(* PLC project Unnamed, Unknown Unnamed 1 *)
(* stored: creationDateTime 2023-01-31T01:35:27, modificationDateTime 2023-04-25T02:26:45 *)

PROGRAM WaterIrrigation
  VAR
    OUTGOING_VALVE AT %QX0.0 : BOOL;
    OUTGOING_PUMP AT %QX0.1 : BOOL;
    INCOMING_PUMP AT %QX0.2 : BOOL;
    TANK_FULL AT %QX0.3 : BOOL;
    PULSE AT %QX0.4 : BOOL;
    TANK_EMPTY AT %QX0.5 : BOOL;
    MANUAL AT %QX0.6 : BOOL;
    PB_INCOMING_OPEN AT %IX0.0 : BOOL;
    PB_INCOMING_CLOSE AT %IX0.1 : BOOL;
    PB_OUTGOING_OPEN AT %IX0.2 : BOOL;
    PB_OUTGOING_CLOSE AT %IX0.3 : BOOL;
    MAX_TANK_LEVEL AT %QW0 : INT := 10;
    TANK_LEVEL_VALUE AT %QW2 : INT := 10;
    WATER_MOISTURE AT %QW3 : INT := 10;
  END_VAR
  VAR
    TON0 : TON;
    TOF0 : TOF;
    CTUD0 : CTUD;
  END_VAR
  VAR  (* added by the conversion: wires and edge detectors of the diagram *)
    R_TRIG1 : R_TRIG;
    R_TRIG2 : R_TRIG;
  END_VAR

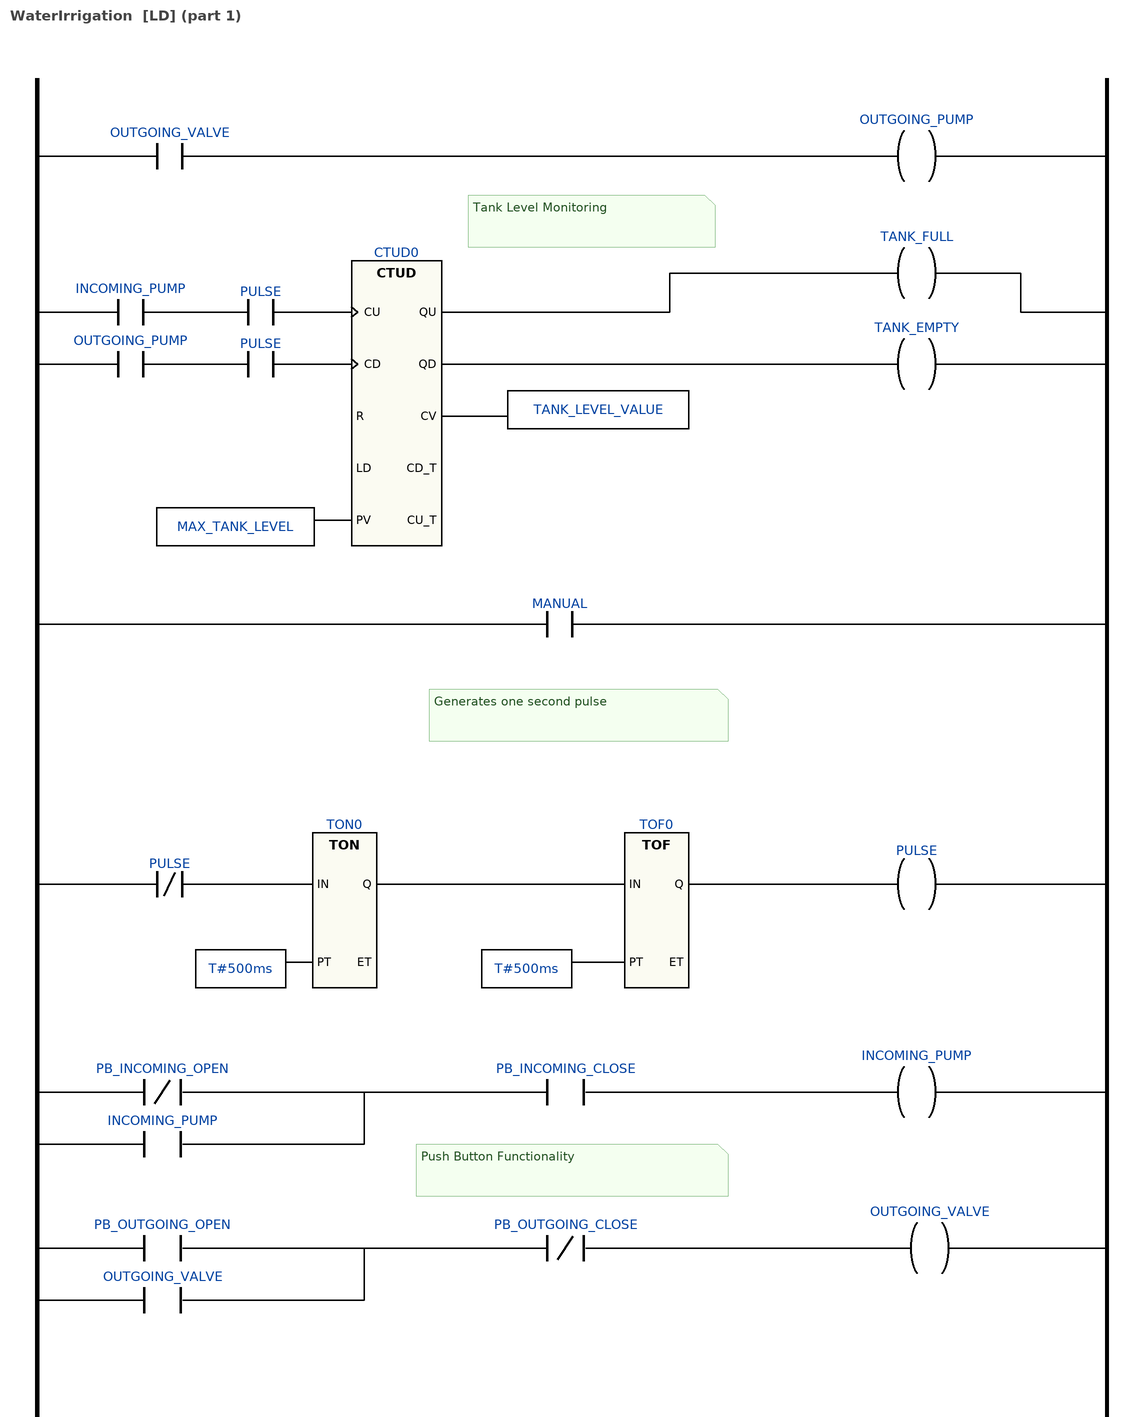
(* LD diagram, written out as Structured Text *)
OUTGOING_PUMP := OUTGOING_VALVE;
(* Tank Level Monitoring *)
R_TRIG1(CLK := INCOMING_PUMP AND PULSE);
R_TRIG2(CLK := OUTGOING_PUMP AND PULSE);
CTUD0(CU := R_TRIG1.Q, CD := R_TRIG2.Q, PV := MAX_TANK_LEVEL);
TANK_FULL := CTUD0.QU;
TANK_EMPTY := CTUD0.QD;
TANK_LEVEL_VALUE := CTUD0.CV;
(* Generates one second pulse *)
TON0(IN := NOT PULSE, PT := T#500ms);
TOF0(IN := TON0.Q, PT := T#500ms);
PULSE := TOF0.Q;
INCOMING_PUMP := (NOT PB_INCOMING_OPEN OR INCOMING_PUMP) AND PB_INCOMING_CLOSE;
(* Push Button Functionality *)
OUTGOING_VALVE := (PB_OUTGOING_OPEN OR OUTGOING_VALVE) AND NOT PB_OUTGOING_CLOSE;
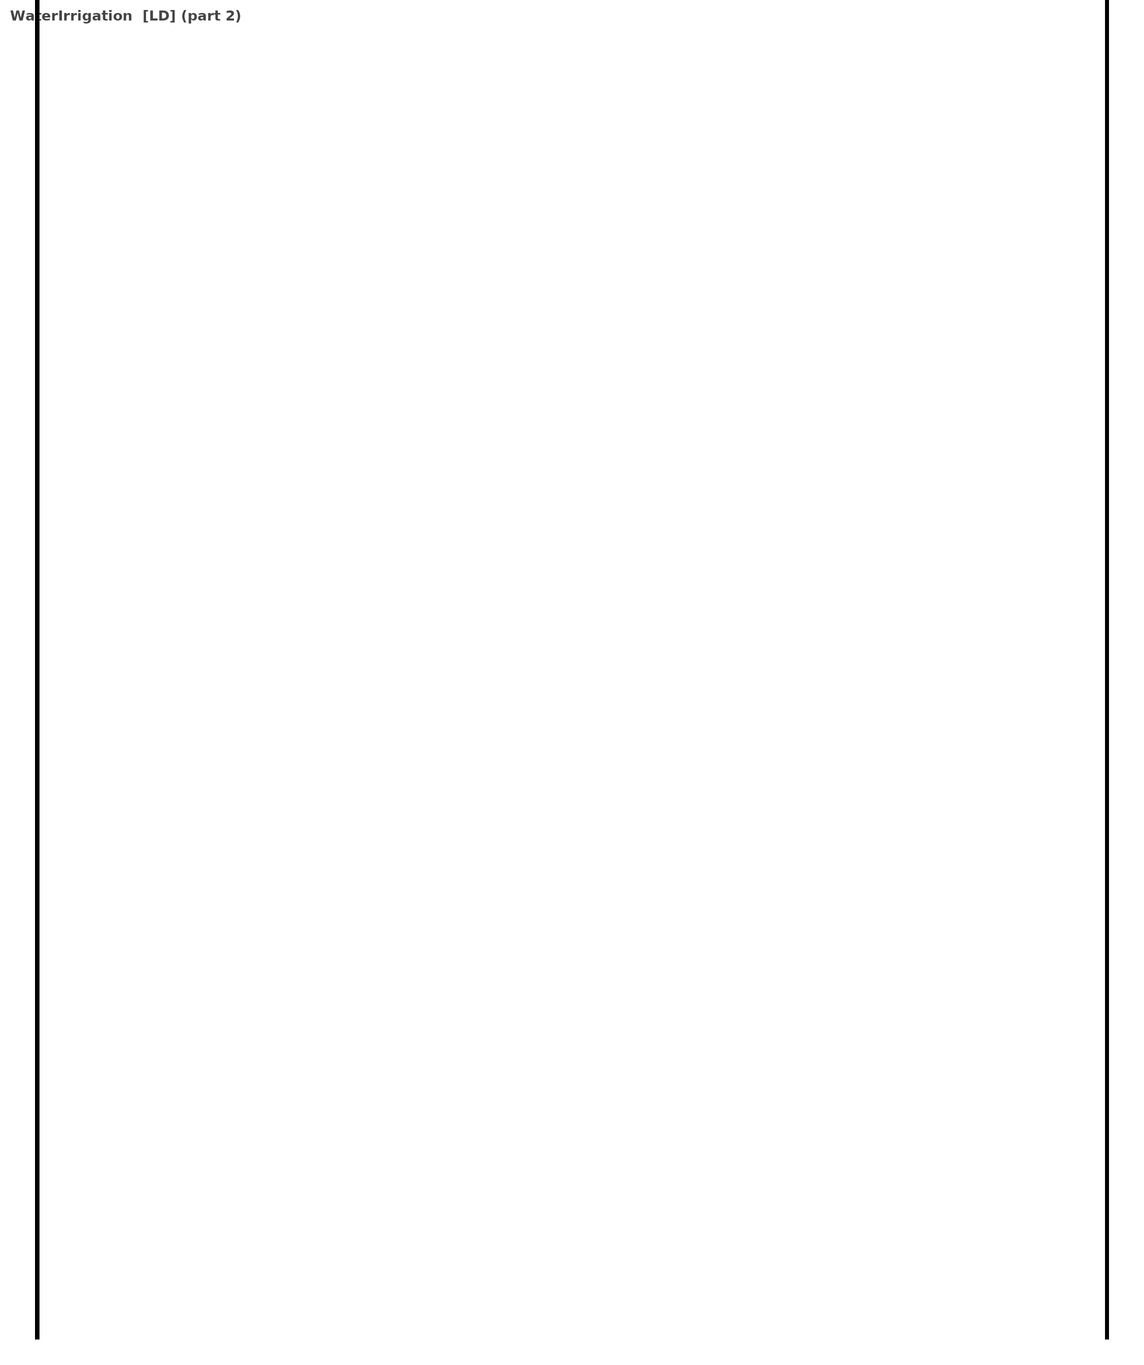
(* drawn but not wired to any output: MANUAL *)
END_PROGRAM

CONFIGURATION Config0
  RESOURCE Res0 ON PLC
    TASK task0(INTERVAL := T#20ms, PRIORITY := 0);
    PROGRAM instance0 WITH task0 : WaterIrrigation;
  END_RESOURCE
END_CONFIGURATION
